PROGRAM MAIN
VAR
END_VAR

END_PROGRAM

(* stored: Version 1.1.0.1
   POU MAIN: Id {acb0024e-8bed-4ca7-9365-fb2f99140800} *)
